FUNCTION_BLOCK FB_PU
VAR_IN_OUT

END_VAR
VAR_INPUT
	Freigabe_auto			: BOOL;
	Freigabe_Deakt_auto		: BOOL;
	Betrieb_Anford_auto		: BOOL;
	Regelung_Modus_auto		: SINT;
	Regelung_Sollw_auto		: REAL;
	Quittierung				: BOOL;
	Parameter_init			: ST_PU_Parameter;
END_VAR
VAR_OUTPUT
	{attribute 'OPC.UA.DA' := '1'}Parameter				: ST_PU_Parameter;			
	{attribute 'OPC.UA.DA' := '1'}Steuerung				: ST_PU_Steuerung;			
	{attribute 'OPC.UA.DA' := '1'}Stellwert				: ST_PU_Stellwert;			
	{attribute 'OPC.UA.DA' := '1'}Zustand					: ST_PU_Zustand;		

END_VAR
VAR
	Zustandscheck			: FB_PU_Zustandscheck;
	Logik					: FB_PU_Logik;
	Ablaufsteuerung			: FB_PU_Ablaufsteuerung;
	Sollwertscheck			: FB_PU_Sollwertscheck;
	Regelung				: FB_PU_Regelung;
	Stellwertscheck			: FB_PU_Stellwertscheck;
	QuitTrig				: FB_SetResetFallTrigger;

	StatusModul1			: DWORD;
	StatusModul2			: DWORD;
	ControlModul1			: DWORD;
	ControlModul2			: DWORD;


	LeseDaten				: FB_PU_Input;
	SchreibeDaten			: FB_PU_Output;
	(*Genibus					: FB_PU_Genibus_old;*)

	IN_StatusModule			AT %I*: ARRAY [0..5] OF USINT;
	IN_Leistung				AT %I*: UDINT;		(* 0..100% *)

	IN_Leistung_elek		AT %I*: UDINT;	(* W *)
	IN_Leistung_therm		AT %I*: UDINT;	(* W *)
	IN_Energie_elek			AT %I*: UDINT;
	IN_Energie_therm		AT %I*: UDINT;
	IN_Volumenstrom			AT %I*: UDINT;
	IN_Volumen				AT %I*: UDINT;
	IN_Temp_intern			AT %I*: REAL;
	IN_Temp_extern			AT %I*: UDINT;
	IN_Temp_elek			AT %I*: UDINT;
	IN_Drehzahl				AT %I*: UDINT;	(* U/min *)
	IN_Frequenz_Motor		AT %I*: UDINT;	(* Hz *)
	IN_Zeit_Betrieb			AT %I*: UDINT;		(* h *)
	IN_Anzahl_Starts		AT %I*: UDINT;
	IN_Modul_Meld_Code1		AT %I*: USINT;
	IN_Modul_Meld_Code2		AT %I*: USINT;
	IN_Druckdifferenz		AT %I*: UDINT;

	IN_Temp_intern_GeniReply	AT %I*: ST_PU_Genibus;
	OUT_Temp_intern_GeniRequest	AT %Q*: ST_PU_Genibus;
	OUT_ControlModule			AT %Q*: ARRAY [0..4] OF USINT;

	Quittierer : BOOL := FALSE;

	Temp_vorl: REAL;
	Genibus: FB_PU_Genibus;
END_VAR

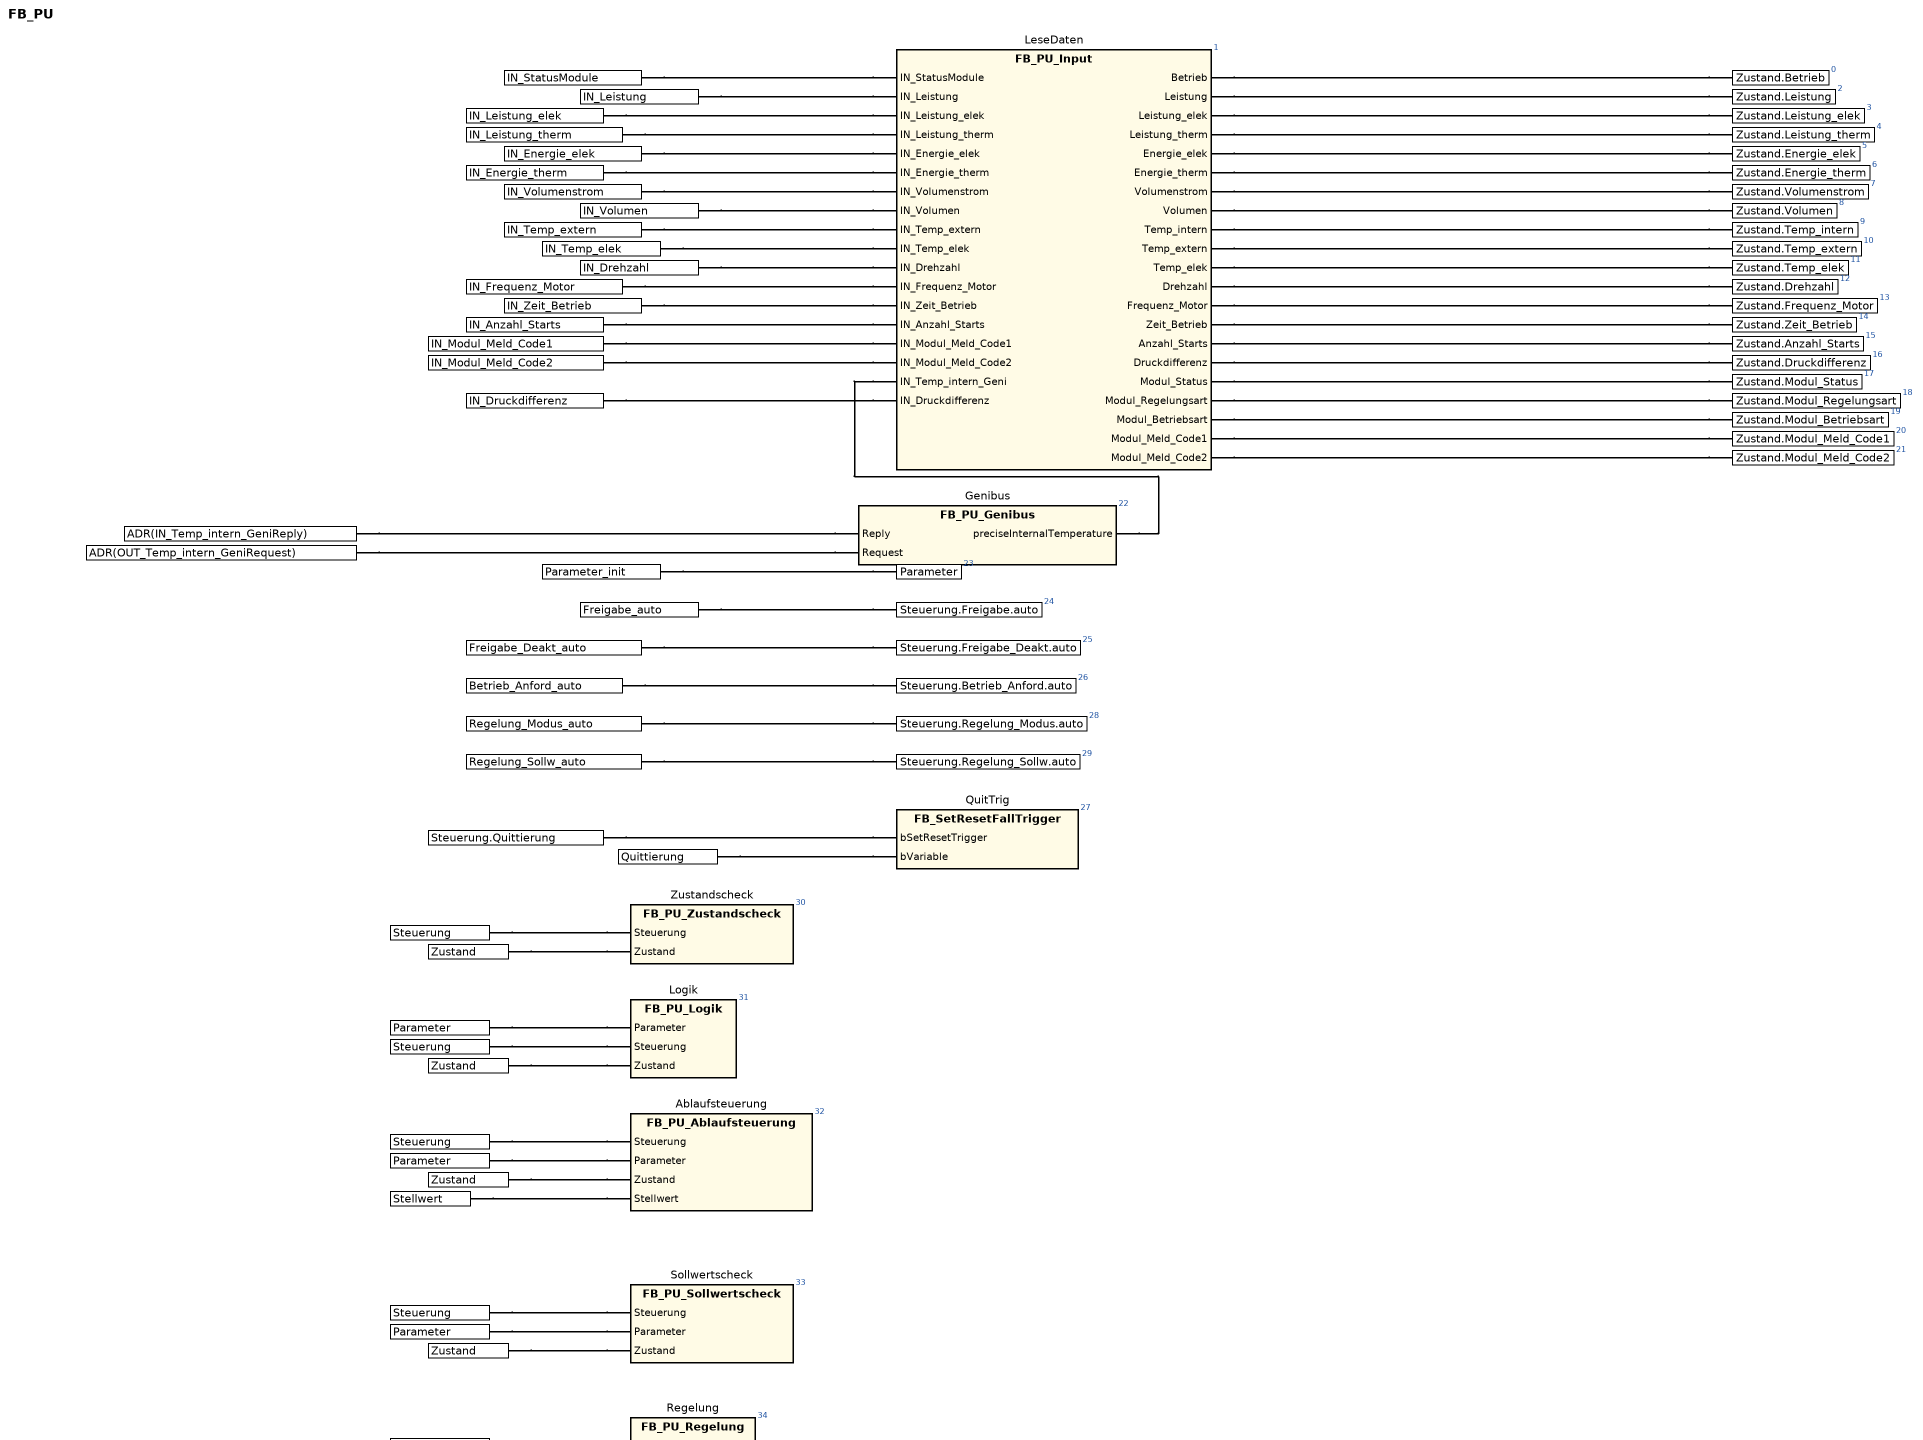
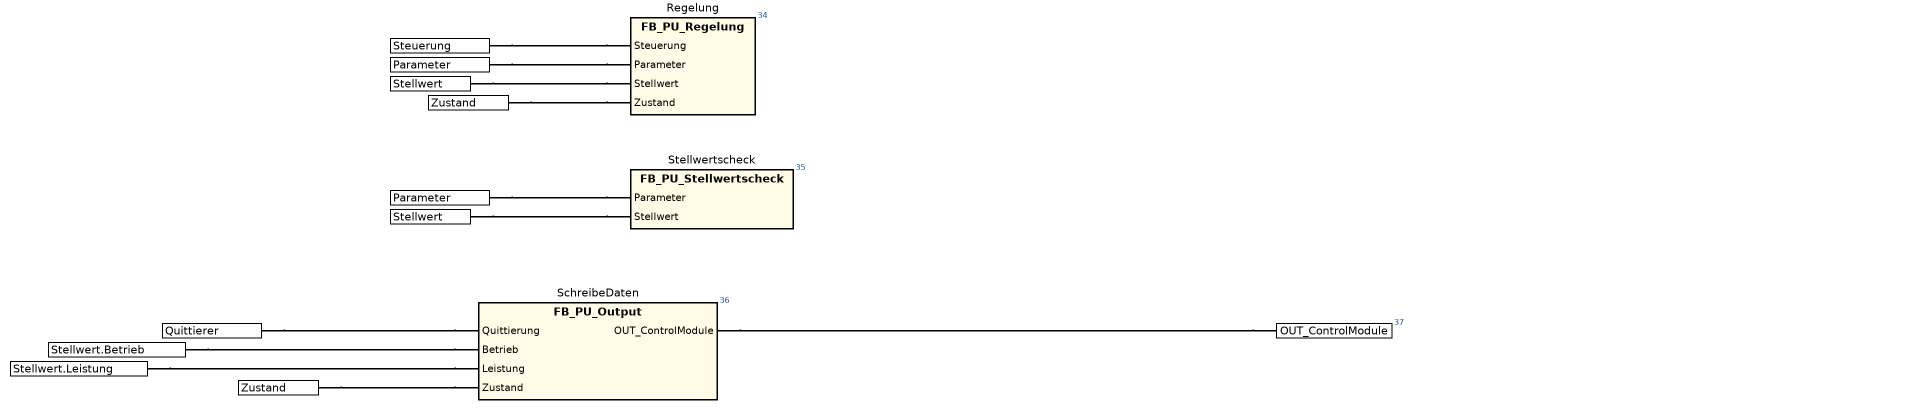
Zustand.Betrieb := LeseDaten.Betrieb;
LeseDaten(
    IN_StatusModule := IN_StatusModule,
    IN_Leistung := IN_Leistung,
    IN_Leistung_elek := IN_Leistung_elek,
    IN_Leistung_therm := IN_Leistung_therm,
    IN_Energie_elek := IN_Energie_elek,
    IN_Energie_therm := IN_Energie_therm,
    IN_Volumenstrom := IN_Volumenstrom,
    IN_Volumen := IN_Volumen,
    IN_Temp_extern := IN_Temp_extern,
    IN_Temp_elek := IN_Temp_elek,
    IN_Drehzahl := IN_Drehzahl,
    IN_Frequenz_Motor := IN_Frequenz_Motor,
    IN_Zeit_Betrieb := IN_Zeit_Betrieb,
    IN_Anzahl_Starts := IN_Anzahl_Starts,
    IN_Modul_Meld_Code1 := IN_Modul_Meld_Code1,
    IN_Modul_Meld_Code2 := IN_Modul_Meld_Code2,
    IN_Temp_intern_Geni := Genibus.preciseInternalTemperature,
    IN_Druckdifferenz := IN_Druckdifferenz); // FB_PU_Input
Zustand.Leistung := LeseDaten.Leistung;
Zustand.Leistung_elek := LeseDaten.Leistung_elek;
Zustand.Leistung_therm := LeseDaten.Leistung_therm;
Zustand.Energie_elek := LeseDaten.Energie_elek;
Zustand.Energie_therm := LeseDaten.Energie_therm;
Zustand.Volumenstrom := LeseDaten.Volumenstrom;
Zustand.Volumen := LeseDaten.Volumen;
Zustand.Temp_intern := LeseDaten.Temp_intern;
Zustand.Temp_extern := LeseDaten.Temp_extern;
Zustand.Temp_elek := LeseDaten.Temp_elek;
Zustand.Drehzahl := LeseDaten.Drehzahl;
Zustand.Frequenz_Motor := LeseDaten.Frequenz_Motor;
Zustand.Zeit_Betrieb := LeseDaten.Zeit_Betrieb;
Zustand.Anzahl_Starts := LeseDaten.Anzahl_Starts;
Zustand.Druckdifferenz := LeseDaten.Druckdifferenz;
Zustand.Modul_Status := LeseDaten.Modul_Status;
Zustand.Modul_Regelungsart := LeseDaten.Modul_Regelungsart;
Zustand.Modul_Betriebsart := LeseDaten.Modul_Betriebsart;
Zustand.Modul_Meld_Code1 := LeseDaten.Modul_Meld_Code1;
Zustand.Modul_Meld_Code2 := LeseDaten.Modul_Meld_Code2;
Genibus(Reply := ADR(IN_Temp_intern_GeniReply), Request := ADR(OUT_Temp_intern_GeniRequest)); // FB_PU_Genibus
Parameter := Parameter_init;
Steuerung.Freigabe.auto := Freigabe_auto;
Steuerung.Freigabe_Deakt.auto := Freigabe_Deakt_auto;
Steuerung.Betrieb_Anford.auto := Betrieb_Anford_auto;
QuitTrig(bSetResetTrigger := Steuerung.Quittierung, bVariable := Quittierung); // FB_SetResetFallTrigger
Steuerung.Regelung_Modus.auto := Regelung_Modus_auto;
Steuerung.Regelung_Sollw.auto := Regelung_Sollw_auto;
Zustandscheck(Steuerung := Steuerung, Zustand := Zustand); // FB_PU_Zustandscheck
Logik(Parameter := Parameter, Steuerung := Steuerung, Zustand := Zustand); // FB_PU_Logik
Ablaufsteuerung(Steuerung := Steuerung, Parameter := Parameter, Zustand := Zustand, Stellwert := Stellwert); // FB_PU_Ablaufsteuerung
Sollwertscheck(Steuerung := Steuerung, Parameter := Parameter, Zustand := Zustand); // FB_PU_Sollwertscheck
Regelung(Steuerung := Steuerung, Parameter := Parameter, Stellwert := Stellwert, Zustand := Zustand); // FB_PU_Regelung
Stellwertscheck(Parameter := Parameter, Stellwert := Stellwert); // FB_PU_Stellwertscheck
SchreibeDaten(
    Quittierung := Quittierer,
    Betrieb := Stellwert.Betrieb,
    Leistung := Stellwert.Leistung,
    Zustand := Zustand); // FB_PU_Output
OUT_ControlModule := SchreibeDaten.OUT_ControlModule;

END_FUNCTION_BLOCK

(* stored: Version 1.1.0.1, ProductVersion 3.1.4024.9
   POU FB_PU: Id {80203938-a863-4867-ac00-236a92fbcb0e}, SpecialFunc None *)
